{attribute 'enable_dynamic_creation'}
FUNCTION_BLOCK FB_FlipTube EXTENDS FB_PieceBase
VAR_INPUT
END_VAR
VAR_OUTPUT
END_VAR
VAR
	bIsOpen : BOOL;
	nTopLevel : DINT;
	nBottomLevel : DINT;	
END_VAR

METHOD FB_init : BOOL
VAR_INPUT
	bInitRetains : BOOL; // if TRUE, the retain variables are initialized (warm start / cold start)
	bInCopyCode : BOOL;  // if TRUE, the instance afterwards gets moved into the copy code (online change)
END_VAR
eObjectType := E_ObjectType.OBJECTTYPE_FlipTube;
eObjectGroup := E_ObjectGroup.OBJECTGROUP_Piece;
END_METHOD

METHOD M_GetAllProps : ERRORID
VAR_INPUT
	refCmdData : REFERENCE TO  ST_CmdData;
END_VAR
SUPER^.M_GetAllProps(refCmdData);
nCurrentPropIndex := nCurrentPropIndex + 1;
refCmdData.n32Data[nCurrentPropIndex] := BOOL_TO_DINT(bIsOpen);
nCurrentPropIndex := nCurrentPropIndex + 1;
refCmdData.n32Data[nCurrentPropIndex] := nTopLevel;
nCurrentPropIndex := nCurrentPropIndex + 1;
refCmdData.n32Data[nCurrentPropIndex] := nBottomLevel;
END_METHOD

{attribute 'object_name' := 'M_SetAllProps'}
METHOD M_SetAllProps : ERRORID
VAR_INPUT
	refCmdData	: REFERENCE TO ST_CmdData;
END_VAR
M_SetAllProps := SUPER^.M_SetAllProps(refCmdData);

IF M_SetAllProps > 0 THEN
	RETURN;
END_IF
nCurrentPropIndex := nCurrentPropIndex + 1;
nSpecPropIndex := nCurrentPropIndex;

bIsOpen := DINT_TO_BOOL(refCmdData.n32Data[nCurrentPropIndex]);
nCurrentPropIndex := nCurrentPropIndex + 1;
nTopLevel := refCmdData.n32Data[nCurrentPropIndex];
nCurrentPropIndex := nCurrentPropIndex + 1;
nBottomLevel := refCmdData.n32Data[nCurrentPropIndex];

nNoOfProps := nCurrentPropIndex + 1;
END_METHOD

METHOD M_SetSingleProp : ERRORID
VAR_INPUT
	refCmdData : REFERENCE TO  ST_CmdData;
END_VAR
IF refCmdData.aHeader[1] = nSpecPropIndex THEN
	bIsOpen := DINT_TO_BOOL(refCmdData.n32Data[0]);
ELSIF refCmdData.aHeader[1] + 1 = nSpecPropIndex THEN
	nTopLevel := refCmdData.n32Data[0];
ELSIF refCmdData.aHeader[1] + 2 = nSpecPropIndex THEN
	nBottomLevel := refCmdData.n32Data[0];
ELSE
	M_SetSingleProp := SUPER^.M_SetSingleProp(refCmdData);
END_IF
END_METHOD

PROPERTY P_bIsOpen : BOOL
GET
P_bIsOpen := bIsOpen;
END_GET
SET
bIsOpen := P_bIsOpen;
END_SET
END_PROPERTY

PROPERTY P_nBottomLevel : DINT
GET
P_nBottomLevel := nBottomLevel;
END_GET
END_PROPERTY

PROPERTY P_nTopLevel : DINT
GET
P_nTopLevel := nTopLevel;
END_GET
END_PROPERTY

END_FUNCTION_BLOCK

(* stored: Version 1.1.0.1, ProductVersion 3.1.4022.18
   POU FB_FlipTube: Id {be527c7b-c7ab-41e5-a0db-9c314abc2e6d}, SpecialFunc None
   Method FB_init: Id {13295405-401f-4229-8512-62ccdd60b0bd}
   Method M_GetAllProps: Id {8632fa0b-f0a1-4150-8497-c788dee95e12}
   Method M_SetAllProps: Id {33418384-c955-4035-8e87-98ac9595dcb1}
   Method M_SetSingleProp: Id {bbe18f58-82d7-425d-a111-e37555db68fe}
   Property P_bIsOpen: Id {cbc33f89-73a1-49de-a2fe-63cc3b4b7670}
   Get Get: Id {9c9795ef-b460-4b31-af27-f59c37b61316}
   Set Set: Id {1afd7639-2b13-4b4d-969c-570270d847f6}
   Property P_nBottomLevel: Id {397dbe44-794d-4344-b75f-544d9a414284}
   Get Get: Id {2af393a1-0490-4c2c-b333-470859f5c842}
   Property P_nTopLevel: Id {0b360c8b-b833-4c6d-9ce5-ab35309ce737}
   Get Get: Id {514acb15-340b-4e28-a4ff-3a8c548fcdb6} *)
